PROGRAM BasicTests
VAR
    Motor: ST_MotionStage;
    fbMotion: FB_MotionStageSim;
    fbRequest: FB_MotionRequest;

    bError: BOOL;
    errState: MC_AxisStates;
END_VAR

fbRequest(stMotionStage := Motor);
fbMotion(stMotionStage := Motor);

CASE Motor.Axis.Status.MotionState OF
   MC_AXISSTATE_ERRORSTOP,
   MC_AXISSTATE_STOPPING,
   MC_AXISSTATE_HOMING,
   MC_AXISSTATE_DISCRETEMOTION,
   MC_AXISSTATE_CONTINOUSMOTION,
   MC_AXISSTATE_SYNCHRONIZEDMOTION:
        IF NOT Motor.bBrakeRelease THEN
            bError := TRUE;
            errState := Motor.Axis.Status.MotionState;
        END_IF
END_CASE

END_PROGRAM

(* stored: Version 1.1.0.1
   POU BasicTests: Id {32c6d46d-3ef9-49e6-91a9-6852b4cc0f44}, SpecialFunc None *)
